TYPE DUT_HMI_04_MANUALS :
STRUCT
	PS : ARRAY[0..CNC.NUM_MAX_MANUALS_04-1] OF BOOL;
	LS : ARRAY[0..CNC.NUM_MAX_MANUALS_04-1] OF BOOL;
END_STRUCT
END_TYPE

(* stored: Version 1.1.0.1, ProductVersion 3.1.4024.13
   DUT DUT_HMI_04_MANUALS: Id {b23a9bed-c741-41c7-8a44-1b99f3e61c2d} *)
